TYPE ST_ExtendedWarnings :
STRUCT
	{attribute 'pytmc' := '
		pv: REM_NOT_POSSIBLE
		io: i
		field: ZNAM OK
		field: ONAM NOT_OK
		field: ZSV NO_ALARM
		field: OSV MINOR
	'}
	bRemoteControlNotPossible: BOOL;
	{attribute 'pytmc' := '
		pv: CTRL_SP_NOT_ALLOWED
		io: i
		field: ZNAM OK
		field: ONAM NOT_OK
		field: ZSV NO_ALARM
		field: OSV MINOR
	'}
	bControlModeSPNotAllowed : BOOL;
	{attribute 'pytmc' := '
		pv: ZERO_STATUS
		io: i
		field: ZNAM ENABLED
		field: ONAM DISABLED
		field: ZSV NO_ALARM
		field: OSV MINOR
	'}
	bZeroDisabled : BOOL;
	{attribute 'pytmc' := '
		pv: PFO_STATUS
		io: i
		field: ZNAM ENABLED
		field: ONAM DISABLED
		field: ZSV NO_ALARM
		field: OSV MINOR
	'}
	bPFODeactivated : BOOL;
	{attribute 'pytmc' := '
		pv: PRES_SP_OOR
		io: i
		field: ZNAM OK
		field: ONAM NOT_OK
		field: ZSV NO_ALARM
		field: OSV MAJOR
	'}
	bPressureSPOutOfRange : BOOL;
	{attribute 'pytmc' := '
		pv: POS_SP_OOR
		io: i
		field: ZNAM OK
		field: ONAM NOT_OK
		field: ZSV NO_ALARM
		field: OSV MAJOR
	'}
	bPositionSPOutOfRange : BOOL;
	{attribute 'pytmc' := '
		pv: CTRL_SP_OOR
		io: i
		field: ZNAM OK
		field: ONAM NOT_OK
		field: ZSV NO_ALARM
		field: OSV MAJOR
	'}
	bCtrlSPOutOfRange : BOOL;
	{attribute 'pytmc' := '
		pv: GENCTRL_SP_OOR
		io: i
		field: ZNAM OK
		field: ONAM NOT_OK
		field: ZSV NO_ALARM
		field: OSV MAJOR
	'}
	bGeneralCtrlSPOutOfRange : BOOL;
	{attribute 'pytmc' := '
		pv: PROC_DATA_NOT_VALID
		io: i
		field: ZNAM OK
		field: ONAM NOT_OK
		field: ZSV NO_ALARM
		field: OSV MAJOR
	'}
	bProcDataSettingsNotvalid : BOOL;
END_STRUCT
END_TYPE

(* stored: Version 1.1.0.1, ProductVersion 3.1.4022.18
   DUT ST_ExtendedWarnings: Id {7b622667-e2e2-4049-b120-661b229c539e} *)
